TYPE ST_FSoE_02Byte :
STRUCT
	CMD		: BYTE;
	SafeData1 	: WORD;
	CRC1		: WORD;
	ConnID		: WORD;
END_STRUCT
END_TYPE

(* stored: Version 1.1.0.1, ProductVersion 3.1.4024.5
   DUT ST_FSoE_02Byte: Id {e6f166e1-e444-493c-8cb4-3fc5fabd9184} *)
